VISUALIZATION Sequencer_Visualization  // 2x2
END_VISUALIZATION

(* stored: Version 1.1.0.1, ProductVersion 3.1.4024.15
   Visu Sequencer_Visualization: Id {70f985d4-413b-46f6-8424-0f3a0c5a4ac2} *)
